Fanuc KAREL source: ka00120.KL

PROGRAM KA00120
%STACKSIZE=65535
%PRIORITY=65535
%NOLOCKGROUP
-- UNRESOLVED DECLARATIONS (source type spelling not recovered)
-- SRC : TYPE_0x001C (type_u16=0x001C)
-- DST : ARRAY[2] OF TYPE_0x0017 (type_u16=0x2017)
BEGIN
-- UNRESOLVED_PC line 7 opcodes [9D 22 A5] marker_code=0
-- UNRESOLVED_PC line 8 opcodes [21 22 9D 33 B4] marker_code=15
END KA00120
